// TIA Portal V16 export
// export: Created 2025-05-24T14:08:02.508149Z, ExportSetting WithDefaults, DisplayName Totally Integrated Automation Portal, DisplayVersion V16, DisplayName TIA Portal Version Control Interface, DisplayVersion V16, DisplayName TIA Portal Openness, DisplayVersion V16, DisplayName STEP 7 Professional, DisplayVersion V16, DisplayName STEP 7 Safety, DisplayVersion V16, DisplayName WinCC Advanced, DisplayVersion V16
DATA_BLOCK "Blinker_BlueConstant"   // DB65
VERSION : 0.1
// stored: AutoNumber true, InstanceOfName Blinker, InstanceOfType FB
"Blinker"
   // VAR_INPUT
   //    Enable : Bool;
   //    BlinkTime : Time;
   // END_VAR
   // VAR_OUTPUT
   //    Q_Blink : Bool;
   //    Q_Blink2 : Bool;
   // END_VAR
   // VAR RETAIN
   //    BlinkTimer : TON;
   // END_VAR
BEGIN
END_DATA_BLOCK
